// Mitsubishi GX Works2 project: pr1   PLC: Q03UDV

PROGRAM MAIN
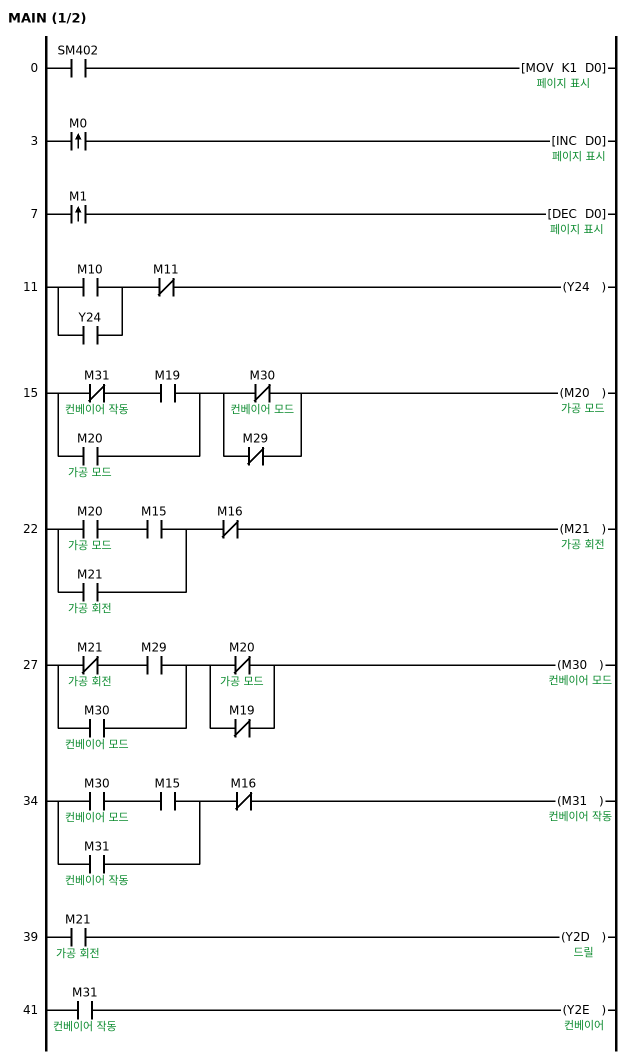
0     LD      SM402
      MOV     K1 D0  ; 페이지 표시
3     LDP     M0
      INC     D0
7     LDP     M1
      DEC     D0
11    LD      M10
      OR      Y24
      ANI     M11
      OUT     Y24
15    LDI     M31  ; 컨베이어 작동
      AND     M19
      OR      M20  ; 가공 모드
      LDI     M30  ; 컨베이어 모드
      ORI     M29
      ANB
      OUT     M20  ; 가공 모드
22    LD      M20  ; 가공 모드
      AND     M15
      OR      M21  ; 가공 회전
      ANI     M16
      OUT     M21  ; 가공 회전
27    LDI     M21  ; 가공 회전
      AND     M29
      OR      M30  ; 컨베이어 모드
      LDI     M20  ; 가공 모드
      ORI     M19
      ANB
      OUT     M30  ; 컨베이어 모드
34    LD      M30  ; 컨베이어 모드
      AND     M15
      OR      M31  ; 컨베이어 작동
      ANI     M16
      OUT     M31  ; 컨베이어 작동
39    LD      M21  ; 가공 회전
      OUT     Y2D  ; 드릴
41    LD      M31  ; 컨베이어 작동
      OUT     Y2E  ; 컨베이어
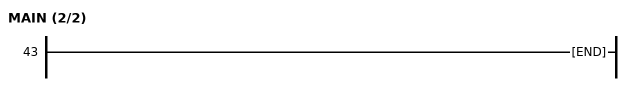
43    END
END_PROGRAM
